(* IEC 61131-3 sources: CannyIEC/extracted_st/library_information/islibreleased, 1 file *)

(* ---- IsLibReleased.st ---- *)
(* --- Interface --- *)
// This function has been automatically generated from the project information.
FUNCTION IsLibReleased : BOOL
VAR_INPUT

END_VAR
(* --- Implementation --- *)
IsLibReleased := FALSE;
